PROGRAM ConductivityCtrl
VAR
END_VAR

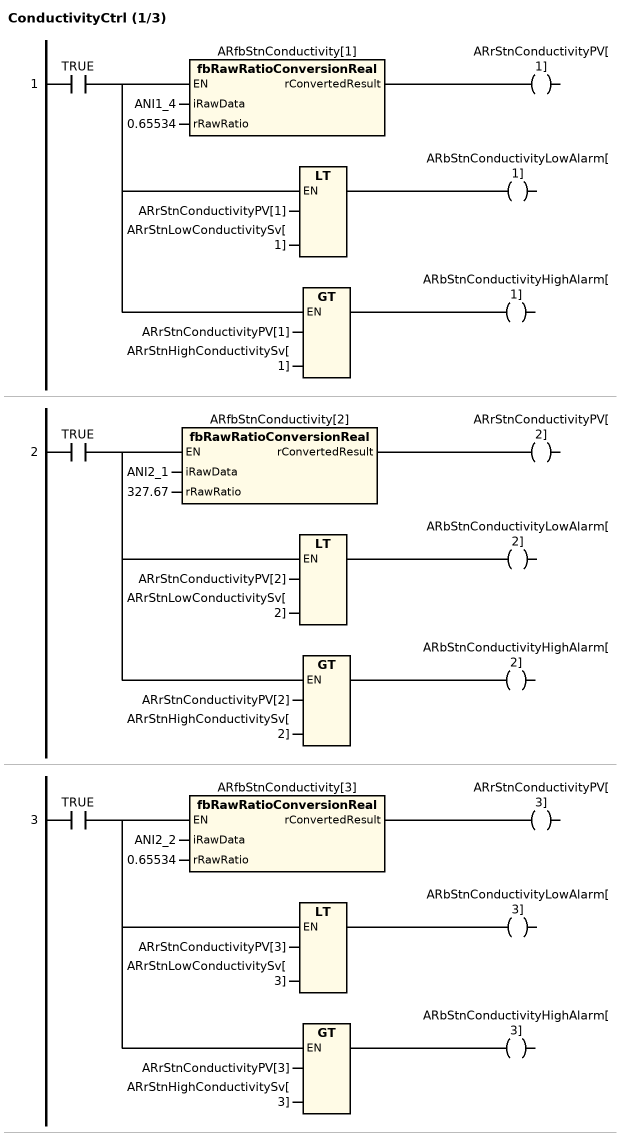
// NETWORK 1
ARfbStnConductivity[1](iRawData := ANI1_4, rRawRatio := 0.65534); // fbRawRatioConversionReal
ARrStnConductivityPV[1] := ARfbStnConductivity[1].rConvertedResult;
ARbStnConductivityLowAlarm[1] := ARrStnConductivityPV[1] < ARrStnLowConductivitySv[1];
ARbStnConductivityHighAlarm[1] := ARrStnConductivityPV[1] > ARrStnHighConductivitySv[1];

// NETWORK 2
ARfbStnConductivity[2](iRawData := ANI2_1, rRawRatio := 327.67); // fbRawRatioConversionReal
ARrStnConductivityPV[2] := ARfbStnConductivity[2].rConvertedResult;
ARbStnConductivityLowAlarm[2] := ARrStnConductivityPV[2] < ARrStnLowConductivitySv[2];
ARbStnConductivityHighAlarm[2] := ARrStnConductivityPV[2] > ARrStnHighConductivitySv[2];

// NETWORK 3
ARfbStnConductivity[3](iRawData := ANI2_2, rRawRatio := 0.65534); // fbRawRatioConversionReal
ARrStnConductivityPV[3] := ARfbStnConductivity[3].rConvertedResult;
ARbStnConductivityLowAlarm[3] := ARrStnConductivityPV[3] < ARrStnLowConductivitySv[3];
ARbStnConductivityHighAlarm[3] := ARrStnConductivityPV[3] > ARrStnHighConductivitySv[3];

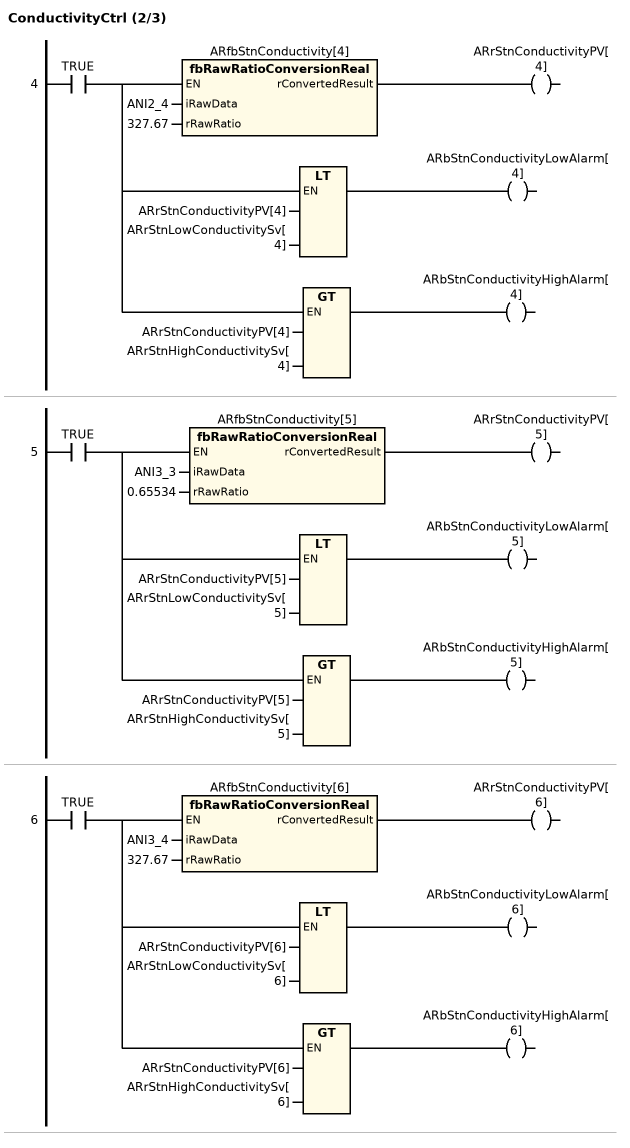
// NETWORK 4
ARfbStnConductivity[4](iRawData := ANI2_4, rRawRatio := 327.67); // fbRawRatioConversionReal
ARrStnConductivityPV[4] := ARfbStnConductivity[4].rConvertedResult;
ARbStnConductivityLowAlarm[4] := ARrStnConductivityPV[4] < ARrStnLowConductivitySv[4];
ARbStnConductivityHighAlarm[4] := ARrStnConductivityPV[4] > ARrStnHighConductivitySv[4];

// NETWORK 5
ARfbStnConductivity[5](iRawData := ANI3_3, rRawRatio := 0.65534); // fbRawRatioConversionReal
ARrStnConductivityPV[5] := ARfbStnConductivity[5].rConvertedResult;
ARbStnConductivityLowAlarm[5] := ARrStnConductivityPV[5] < ARrStnLowConductivitySv[5];
ARbStnConductivityHighAlarm[5] := ARrStnConductivityPV[5] > ARrStnHighConductivitySv[5];

// NETWORK 6
ARfbStnConductivity[6](iRawData := ANI3_4, rRawRatio := 327.67); // fbRawRatioConversionReal
ARrStnConductivityPV[6] := ARfbStnConductivity[6].rConvertedResult;
ARbStnConductivityLowAlarm[6] := ARrStnConductivityPV[6] < ARrStnLowConductivitySv[6];
ARbStnConductivityHighAlarm[6] := ARrStnConductivityPV[6] > ARrStnHighConductivitySv[6];

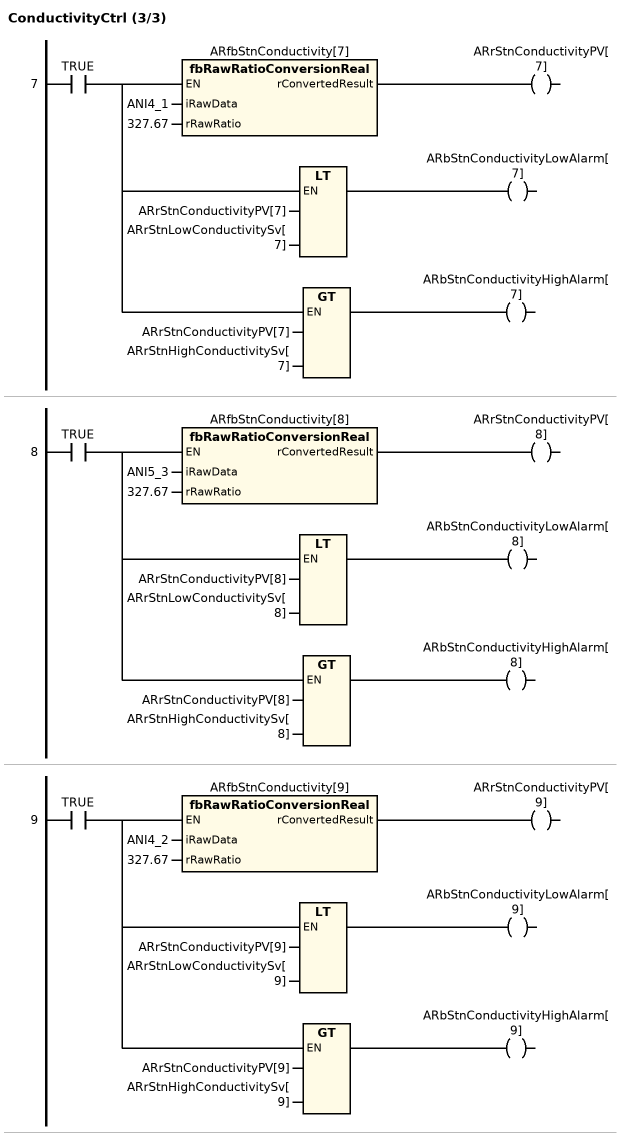
// NETWORK 7
ARfbStnConductivity[7](iRawData := ANI4_1, rRawRatio := 327.67); // fbRawRatioConversionReal
ARrStnConductivityPV[7] := ARfbStnConductivity[7].rConvertedResult;
ARbStnConductivityLowAlarm[7] := ARrStnConductivityPV[7] < ARrStnLowConductivitySv[7];
ARbStnConductivityHighAlarm[7] := ARrStnConductivityPV[7] > ARrStnHighConductivitySv[7];

// NETWORK 8
ARfbStnConductivity[8](iRawData := ANI5_3, rRawRatio := 327.67); // fbRawRatioConversionReal
ARrStnConductivityPV[8] := ARfbStnConductivity[8].rConvertedResult;
ARbStnConductivityLowAlarm[8] := ARrStnConductivityPV[8] < ARrStnLowConductivitySv[8];
ARbStnConductivityHighAlarm[8] := ARrStnConductivityPV[8] > ARrStnHighConductivitySv[8];

// NETWORK 9
ARfbStnConductivity[9](iRawData := ANI4_2, rRawRatio := 327.67); // fbRawRatioConversionReal
ARrStnConductivityPV[9] := ARfbStnConductivity[9].rConvertedResult;
ARbStnConductivityLowAlarm[9] := ARrStnConductivityPV[9] < ARrStnLowConductivitySv[9];
ARbStnConductivityHighAlarm[9] := ARrStnConductivityPV[9] > ARrStnHighConductivitySv[9];

END_PROGRAM

(* stored: Version 1.1.0.1, ProductVersion 3.1.4024.12
   POU ConductivityCtrl: Id {550d10c2-099d-44b9-b12c-ab5131615837}, SpecialFunc None *)
